PROGRAM prgReadTextList
VAR_INPUT
END_VAR
VAR_OUTPUT
END_VAR
VAR
	starttt: BOOL;
	readMC_Alarms: FB_ReadTextList;
	readMC_Prompts: FB_ReadTextList;
	readMC_Warnings: FB_ReadTextList;
	resett: BOOL;
	readS1_Alarms: FB_ReadTextList;
	readS1_Prompts: FB_ReadTextList;
	readS1_Warnings: FB_ReadTextList;
	
	readS2_Alarms: FB_ReadTextList;
	readS2_Prompts: FB_ReadTextList;
	readS2_Warnings: FB_ReadTextList;
	
	readS3_Alarms: FB_ReadTextList;
	readS3_Prompts: FB_ReadTextList;
	readS3_Warnings: FB_ReadTextList;
	
	readS4_Alarms: FB_ReadTextList;
	readS4_Prompts: FB_ReadTextList;
	readS4_Warnings: FB_ReadTextList;
	
	readS5_Alarms: FB_ReadTextList;
	readS5_Prompts: FB_ReadTextList;
	readS5_Warnings: FB_ReadTextList;
	
	readS6_Alarms: FB_ReadTextList;
	readS6_Prompts: FB_ReadTextList;
	readS6_Warnings: FB_ReadTextList;
	
	

	
END_VAR
VAR // added by the converter: edge detectors and wires of the graphical bodies
    _rt1, _rt2, _rt3, _rt4 : R_TRIG;
END_VAR

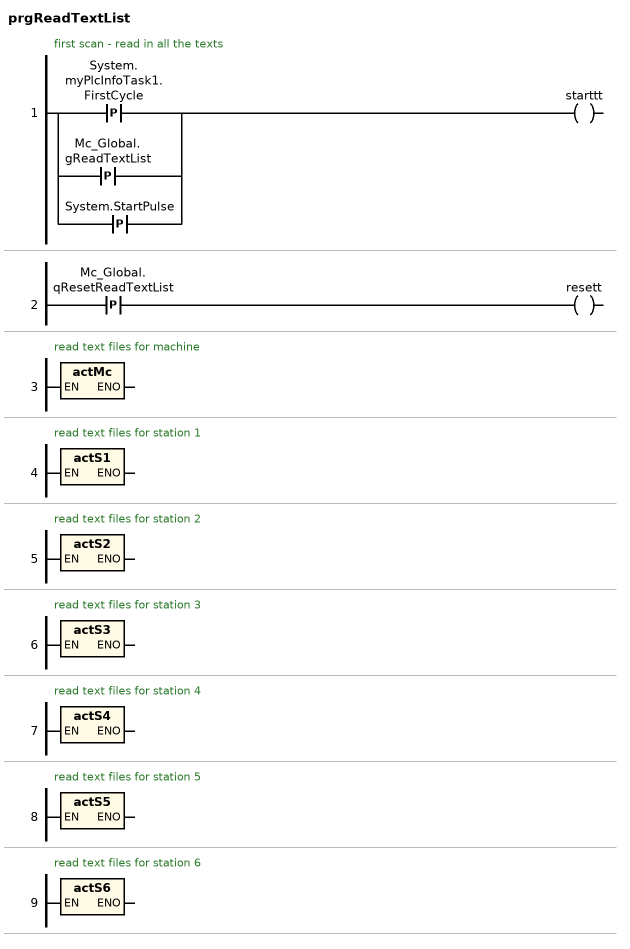
// NETWORK 1
// first scan - read in all the texts
_rt1(CLK := System.myPlcInfoTask1.FirstCycle);
_rt2(CLK := Mc_Global.gReadTextList);
_rt3(CLK := System.StartPulse);
starttt := _rt1.Q OR _rt2.Q OR _rt3.Q;

// NETWORK 2
_rt4(CLK := Mc_Global.qResetReadTextList);
resett := _rt4.Q;

// NETWORK 3
// read text files for machine
actMc();

// NETWORK 4
// read text files for station 1
actS1();

// NETWORK 5
// read text files for station 2
actS2();

// NETWORK 6
// read text files for station 3
actS3();

// NETWORK 7
// read text files for station 4
actS4();

// NETWORK 8
// read text files for station 5
actS5();

// NETWORK 9
// read text files for station 6
actS6();

ACTION actMc:
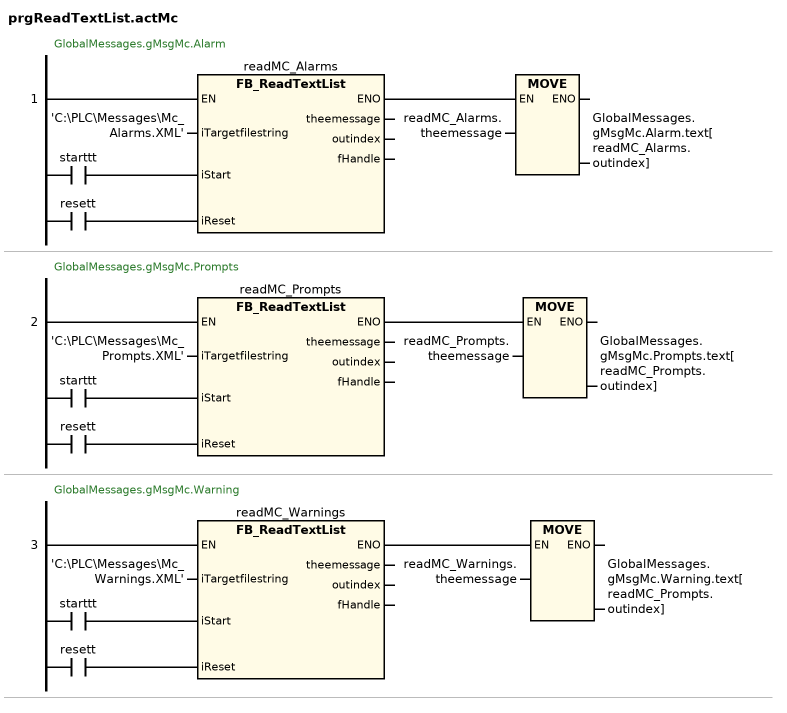
// NETWORK 1
// GlobalMessages.gMsgMc.Alarm
readMC_Alarms(iTargetfilestring := 'C:\PLC\Messages\Mc_Alarms.XML', iStart := starttt, iReset := resett); // FB_ReadTextList
GlobalMessages.gMsgMc.Alarm.text[readMC_Alarms.outindex] := readMC_Alarms.theemessage;

// NETWORK 2
// GlobalMessages.gMsgMc.Prompts
readMC_Prompts(iTargetfilestring := 'C:\PLC\Messages\Mc_Prompts.XML', iStart := starttt, iReset := resett); // FB_ReadTextList
GlobalMessages.gMsgMc.Prompts.text[readMC_Prompts.outindex] := readMC_Prompts.theemessage;

// NETWORK 3
// GlobalMessages.gMsgMc.Warning
readMC_Warnings(iTargetfilestring := 'C:\PLC\Messages\Mc_Warnings.XML', iStart := starttt, iReset := resett); // FB_ReadTextList
GlobalMessages.gMsgMc.Warning.text[readMC_Prompts.outindex] := readMC_Warnings.theemessage;
END_ACTION

ACTION actS1:
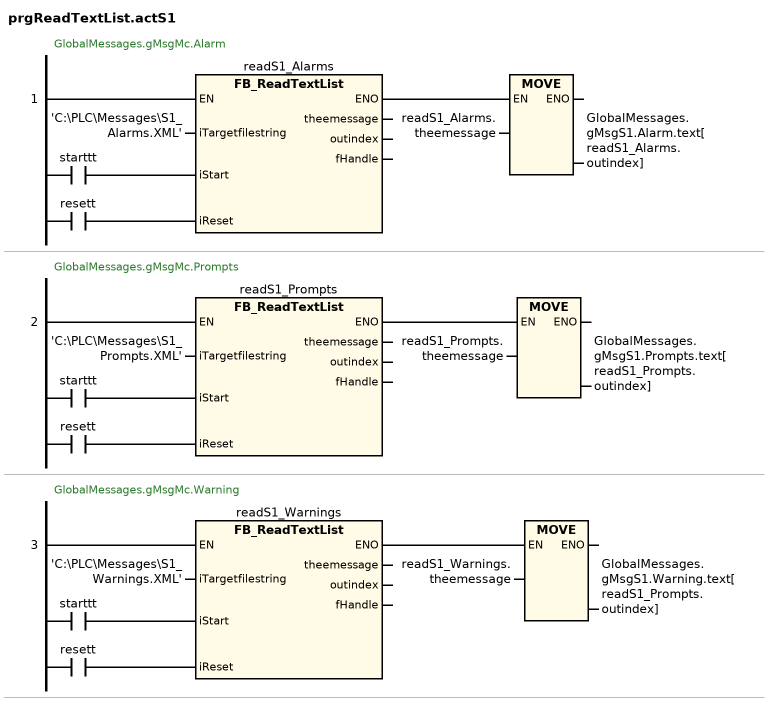
// NETWORK 1
// GlobalMessages.gMsgMc.Alarm
readS1_Alarms(iTargetfilestring := 'C:\PLC\Messages\S1_Alarms.XML', iStart := starttt, iReset := resett); // FB_ReadTextList
GlobalMessages.gMsgS1.Alarm.text[readS1_Alarms.outindex] := readS1_Alarms.theemessage;

// NETWORK 2
// GlobalMessages.gMsgMc.Prompts
readS1_Prompts(iTargetfilestring := 'C:\PLC\Messages\S1_Prompts.XML', iStart := starttt, iReset := resett); // FB_ReadTextList
GlobalMessages.gMsgS1.Prompts.text[readS1_Prompts.outindex] := readS1_Prompts.theemessage;

// NETWORK 3
// GlobalMessages.gMsgMc.Warning
readS1_Warnings(iTargetfilestring := 'C:\PLC\Messages\S1_Warnings.XML', iStart := starttt, iReset := resett); // FB_ReadTextList
GlobalMessages.gMsgS1.Warning.text[readS1_Prompts.outindex] := readS1_Warnings.theemessage;
END_ACTION

ACTION actS2:
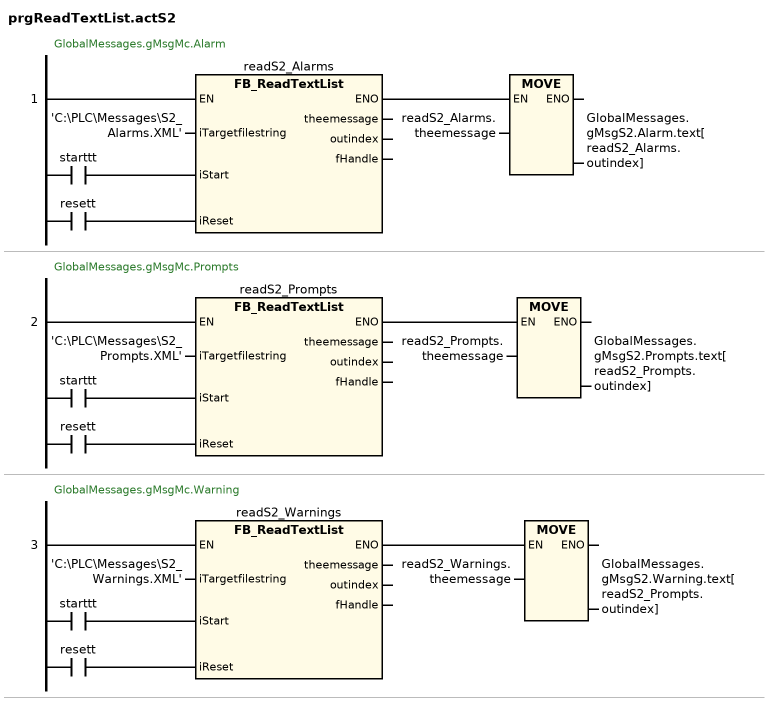
// NETWORK 1
// GlobalMessages.gMsgMc.Alarm
readS2_Alarms(iTargetfilestring := 'C:\PLC\Messages\S2_Alarms.XML', iStart := starttt, iReset := resett); // FB_ReadTextList
GlobalMessages.gMsgS2.Alarm.text[readS2_Alarms.outindex] := readS2_Alarms.theemessage;

// NETWORK 2
// GlobalMessages.gMsgMc.Prompts
readS2_Prompts(iTargetfilestring := 'C:\PLC\Messages\S2_Prompts.XML', iStart := starttt, iReset := resett); // FB_ReadTextList
GlobalMessages.gMsgS2.Prompts.text[readS2_Prompts.outindex] := readS2_Prompts.theemessage;

// NETWORK 3
// GlobalMessages.gMsgMc.Warning
readS2_Warnings(iTargetfilestring := 'C:\PLC\Messages\S2_Warnings.XML', iStart := starttt, iReset := resett); // FB_ReadTextList
GlobalMessages.gMsgS2.Warning.text[readS2_Prompts.outindex] := readS2_Warnings.theemessage;
END_ACTION

ACTION actS3:
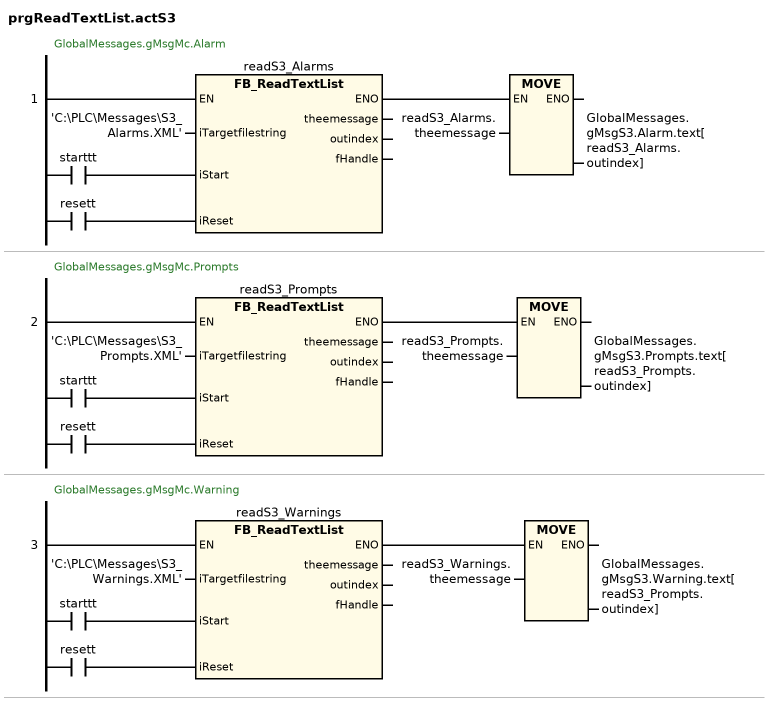
// NETWORK 1
// GlobalMessages.gMsgMc.Alarm
readS3_Alarms(iTargetfilestring := 'C:\PLC\Messages\S3_Alarms.XML', iStart := starttt, iReset := resett); // FB_ReadTextList
GlobalMessages.gMsgS3.Alarm.text[readS3_Alarms.outindex] := readS3_Alarms.theemessage;

// NETWORK 2
// GlobalMessages.gMsgMc.Prompts
readS3_Prompts(iTargetfilestring := 'C:\PLC\Messages\S3_Prompts.XML', iStart := starttt, iReset := resett); // FB_ReadTextList
GlobalMessages.gMsgS3.Prompts.text[readS3_Prompts.outindex] := readS3_Prompts.theemessage;

// NETWORK 3
// GlobalMessages.gMsgMc.Warning
readS3_Warnings(iTargetfilestring := 'C:\PLC\Messages\S3_Warnings.XML', iStart := starttt, iReset := resett); // FB_ReadTextList
GlobalMessages.gMsgS3.Warning.text[readS3_Prompts.outindex] := readS3_Warnings.theemessage;
END_ACTION

ACTION actS4:
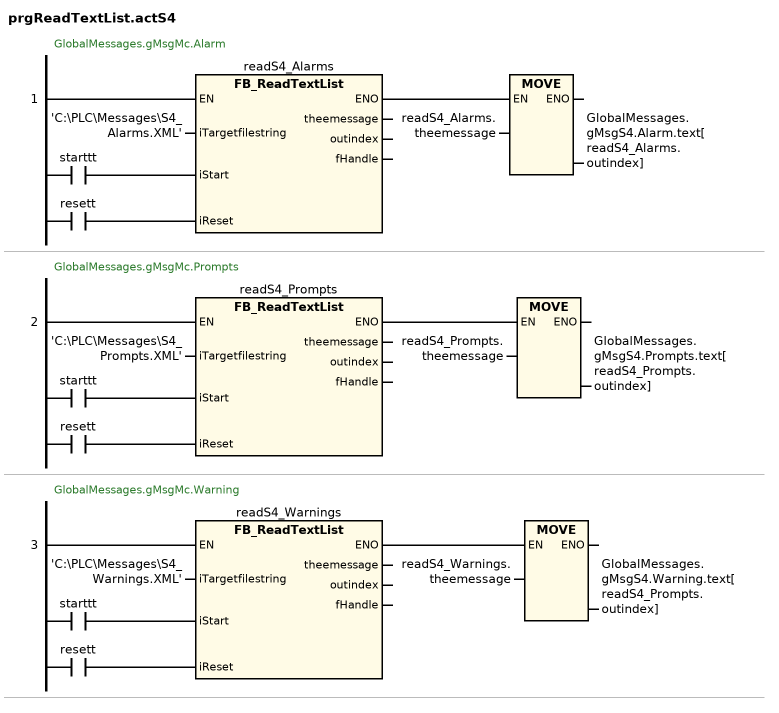
// NETWORK 1
// GlobalMessages.gMsgMc.Alarm
readS4_Alarms(iTargetfilestring := 'C:\PLC\Messages\S4_Alarms.XML', iStart := starttt, iReset := resett); // FB_ReadTextList
GlobalMessages.gMsgS4.Alarm.text[readS4_Alarms.outindex] := readS4_Alarms.theemessage;

// NETWORK 2
// GlobalMessages.gMsgMc.Prompts
readS4_Prompts(iTargetfilestring := 'C:\PLC\Messages\S4_Prompts.XML', iStart := starttt, iReset := resett); // FB_ReadTextList
GlobalMessages.gMsgS4.Prompts.text[readS4_Prompts.outindex] := readS4_Prompts.theemessage;

// NETWORK 3
// GlobalMessages.gMsgMc.Warning
readS4_Warnings(iTargetfilestring := 'C:\PLC\Messages\S4_Warnings.XML', iStart := starttt, iReset := resett); // FB_ReadTextList
GlobalMessages.gMsgS4.Warning.text[readS4_Prompts.outindex] := readS4_Warnings.theemessage;
END_ACTION

ACTION actS5:
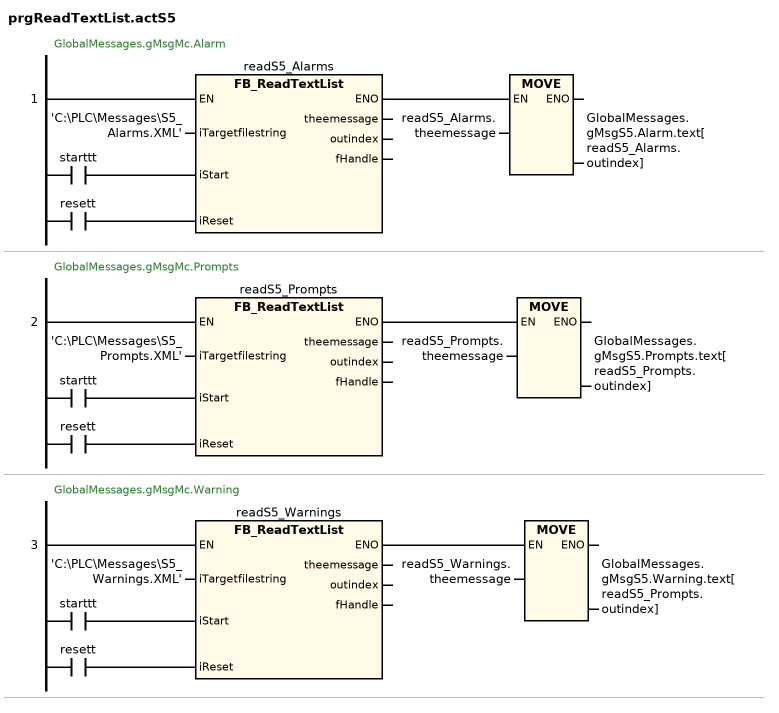
// NETWORK 1
// GlobalMessages.gMsgMc.Alarm
readS5_Alarms(iTargetfilestring := 'C:\PLC\Messages\S5_Alarms.XML', iStart := starttt, iReset := resett); // FB_ReadTextList
GlobalMessages.gMsgS5.Alarm.text[readS5_Alarms.outindex] := readS5_Alarms.theemessage;

// NETWORK 2
// GlobalMessages.gMsgMc.Prompts
readS5_Prompts(iTargetfilestring := 'C:\PLC\Messages\S5_Prompts.XML', iStart := starttt, iReset := resett); // FB_ReadTextList
GlobalMessages.gMsgS5.Prompts.text[readS5_Prompts.outindex] := readS5_Prompts.theemessage;

// NETWORK 3
// GlobalMessages.gMsgMc.Warning
readS5_Warnings(iTargetfilestring := 'C:\PLC\Messages\S5_Warnings.XML', iStart := starttt, iReset := resett); // FB_ReadTextList
GlobalMessages.gMsgS5.Warning.text[readS5_Prompts.outindex] := readS5_Warnings.theemessage;
END_ACTION

ACTION actS6:
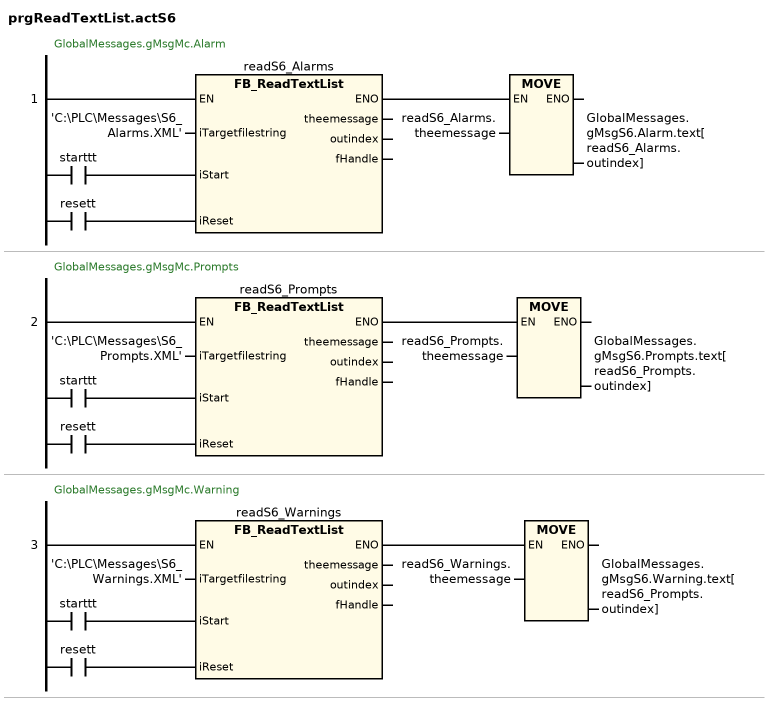
// NETWORK 1
// GlobalMessages.gMsgMc.Alarm
readS6_Alarms(iTargetfilestring := 'C:\PLC\Messages\S6_Alarms.XML', iStart := starttt, iReset := resett); // FB_ReadTextList
GlobalMessages.gMsgS6.Alarm.text[readS6_Alarms.outindex] := readS6_Alarms.theemessage;

// NETWORK 2
// GlobalMessages.gMsgMc.Prompts
readS6_Prompts(iTargetfilestring := 'C:\PLC\Messages\S6_Prompts.XML', iStart := starttt, iReset := resett); // FB_ReadTextList
GlobalMessages.gMsgS6.Prompts.text[readS6_Prompts.outindex] := readS6_Prompts.theemessage;

// NETWORK 3
// GlobalMessages.gMsgMc.Warning
readS6_Warnings(iTargetfilestring := 'C:\PLC\Messages\S6_Warnings.XML', iStart := starttt, iReset := resett); // FB_ReadTextList
GlobalMessages.gMsgS6.Warning.text[readS6_Prompts.outindex] := readS6_Warnings.theemessage;
END_ACTION

END_PROGRAM

(* stored: Version 1.1.0.1, ProductVersion 3.1.4024.11
   POU prgReadTextList: Id {d6a5149c-50b0-4a11-a582-a620d2c47288}, SpecialFunc None
   Action actMc: Id {157a6c63-6d4c-45c6-8dc8-3c144652a0e7}
   Action actS1: Id {a7440002-b0d2-4e88-a517-f381ecc90d05}
   Action actS2: Id {13b49868-b77c-4046-a934-60c3f5a31408}
   Action actS3: Id {4d8e9f34-793f-4a49-93fc-660210bb4717}
   Action actS4: Id {115fe2e9-f9a5-4fee-9e84-cb82209a3a44}
   Action actS5: Id {264875e7-df4b-44b6-b3da-59ea07f855f6}
   Action actS6: Id {c1f80be3-3b0e-4d50-9a5d-77daa2e60c56} *)
